Fanuc KAREL source: foo.kl

PROGRAM foo
%ALPHABETIZE
%COMMENT = ''
%NOBUSYLAMP
%NOLOCKGROUP
%NOPAUSE = COMMAND + TPENABLE + ERROR

%INCLUDE lib_a\a.th

%INCLUDE klrdutil


BEGIN
END foo
